FUNCTION_BLOCK FB_Beckhoff_Auxilary
VAR_INPUT
END_VAR
VAR_OUTPUT
END_VAR
VAR
END_VAR

END_FUNCTION_BLOCK

(* stored: Version 1.1.0.1, ProductVersion 3.1.4022.18
   POU FB_Beckhoff_Auxilary: Id {eb9110a2-3fe1-44c4-92a8-343f88ed7467}, SpecialFunc None
   Folder Methods: Id {2ca2faa1-95cb-45f3-ab61-0b9a77bae127}
   Folder Properties: Id {f0043917-6eb3-4dc8-8615-ec2ad0647ca9} *)
